// TwinCAT 3 PLC project PLC1
// ProgramVersion: 3.1.4023.0
// libraries:
//   Tc2_MC2, * (Beckhoff Automation GmbH)
//   Tc2_Standard, * (Beckhoff Automation GmbH)
//   Tc2_System, * (Beckhoff Automation GmbH)
//   Tc3_Module, * (Beckhoff Automation GmbH)
// project tree:
//   / PlcTask.TcTTO
//   POUs/ MAIN.TcPOU
// real-time tasks:
//   TASK PlcTask: cycle T#10ms, priority 20, ADS port 350
// motion (NC):
//   TASK NC-Task 1 SAF: cycle T#2ms, priority 4, ADS port 501
//   TASK NC-Task 1 SVB: cycle T#10ms, priority 8, ADS port 511
//   AXIS Axis 1 (id 1)
//     OtherSettings: AllowMotionCmdToSlave=true
//     encoder EncType=1
//     drive DrvType=5
//       Analog: TorqueSetpointScale=10, ScaleFactorActTorque=0.1
//       TimeComp: TaskDelayCycles=1
//     controller CtrType=1
//       CtrPara: PriorControlFactor=1
//         Observer: BandWidth=20
// variable links:
//   PLC1/PLC1 Instance <-> NC-Task 1 SAF/Axes/Axis 1
//     PlcTask Inputs/MAIN.Axis.NcToPlc <-> Outputs/ToPlc
//     PlcTask Outputs/MAIN.Axis.PlcToNc <-> Inputs/FromPlc

CONFIGURATION PLC1
    RESOURCE PLC ON TwinCAT3
        TASK PlcTask(INTERVAL := T#10ms, PRIORITY := 20);
        PROGRAM MAIN WITH PlcTask : MAIN;
    END_RESOURCE
END_CONFIGURATION

// ---- POUs/MAIN.TcPOU
PROGRAM MAIN
VAR
	
	Axis: AXIS_REF;
	Axis_Enable : MC_Power;
	
	Axis_ReadRefVelocity 	: MC_ReadParameter; // reads Ref Velocity
	totalControlOutput 		: LREAL;
	Jog						: MC_Jog;
	Velocity 				: LREAL := 2000;
	Forward : BOOL;
	Backward : BOOL;
	
	ActVel: LREAL;

END_VAR

Axis_Enable(Axis := Axis, Enable := TRUE, Enable_Positive := TRUE, Enable_Negative := TRUE);


Axis_ReadRefVelocity(
	Axis := Axis, 
	Enable := TRUE, 
	ParameterNumber := MC_AxisParameter.AxisRefVeloOnRefOutput,
	ReadMode := E_ReadMode.READMODE_CYCLIC
);

	// On first cycle RefVelocity reads as 0. Use SEL to NOT divide by 0
totalControlOutput := SEL(Axis_ReadRefVelocity.Value > 0.0 , 0.0 ,Axis.NcToPlc.ActVelo/Axis_ReadRefVelocity.Value*100);

ActVel := Axis.NcToPlc.ActVelo;


Jog(
	Axis:= Axis, 
	JogForward:= Forward, 
	JogBackwards:= Backward, 
	Mode:= MC_JOGMODE_CONTINOUS, 
	Position:= , 
	Velocity:= Velocity, 
	Acceleration:= 1000, 
	Deceleration:= 1000, 
	Jerk:= , 
	Done=> , 
	Busy=> , 
	Active=> , 
	CommandAborted=> , 
	Error=> , 
	ErrorID=> 
);

END_PROGRAM
